# EPICS substitutions: viocs/tb_ps/tb_psApp/Db/septa.substitutions
file "db/septa.db" {
    pattern { family, pos }
        { "SEPTUMINJ", "05" }
}
